PROGRAM P_ADS_1
VAR
	sTextAlarm1				: WSTRING(255);
	sTextAlarm2				: WSTRING(255);
	sTextAlarm3				: WSTRING(255);
	user					: WSTRING(80);
	iNumberAlarm			: INT;
	bTrigger				: BOOL;
	
	fbRead_1: FB_ReadAdsSymByName;
	fbRead_2: FB_ReadAdsSymByName;
	fbRead_3: FB_ReadAdsSymByName;
	fbCyclicReadout: TON;
	fbRead_4: FB_ReadAdsSymByName;
	fbRead_5: FB_ReadAdsSymByName;
	fbLocaltime: FB_LocalSystemTime;

END_VAR

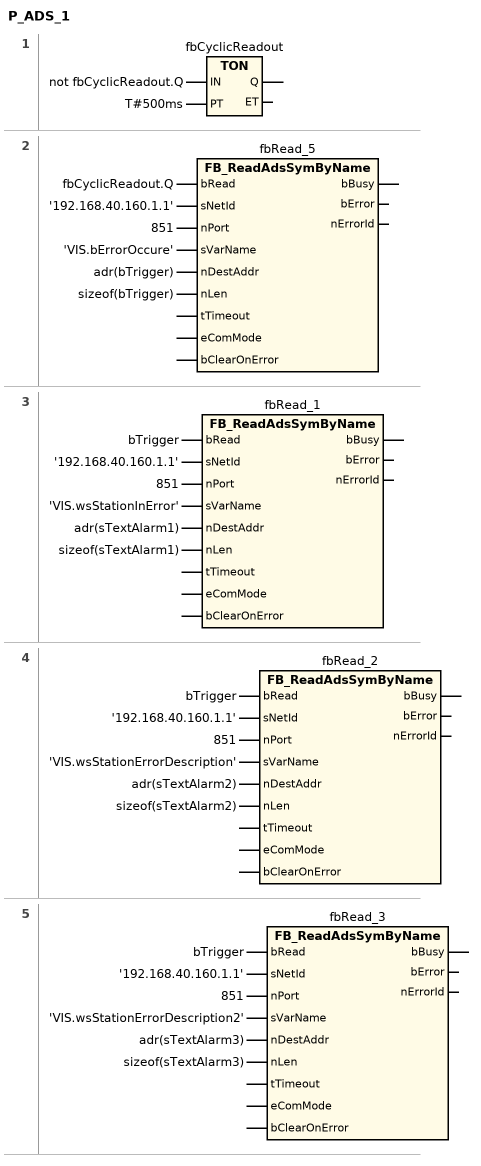
// NETWORK 1
fbCyclicReadout(IN := not fbCyclicReadout.Q, PT := T#500ms); // TON

// NETWORK 2
fbRead_5(
    bRead := fbCyclicReadout.Q,
    sNetId := '192.168.40.160.1.1',
    nPort := 851,
    sVarName := 'VIS.bErrorOccure',
    nDestAddr := adr(bTrigger),
    nLen := sizeof(bTrigger)); // FB_ReadAdsSymByName

// NETWORK 3
fbRead_1(
    bRead := bTrigger,
    sNetId := '192.168.40.160.1.1',
    nPort := 851,
    sVarName := 'VIS.wsStationInError',
    nDestAddr := adr(sTextAlarm1),
    nLen := sizeof(sTextAlarm1)); // FB_ReadAdsSymByName

// NETWORK 4
fbRead_2(
    bRead := bTrigger,
    sNetId := '192.168.40.160.1.1',
    nPort := 851,
    sVarName := 'VIS.wsStationErrorDescription',
    nDestAddr := adr(sTextAlarm2),
    nLen := sizeof(sTextAlarm2)); // FB_ReadAdsSymByName

// NETWORK 5
fbRead_3(
    bRead := bTrigger,
    sNetId := '192.168.40.160.1.1',
    nPort := 851,
    sVarName := 'VIS.wsStationErrorDescription2',
    nDestAddr := adr(sTextAlarm3),
    nLen := sizeof(sTextAlarm3)); // FB_ReadAdsSymByName

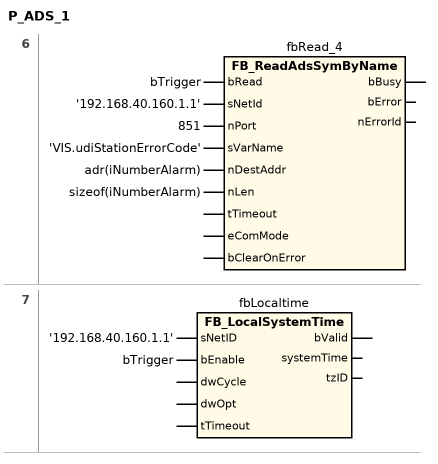
// NETWORK 6
fbRead_4(
    bRead := bTrigger,
    sNetId := '192.168.40.160.1.1',
    nPort := 851,
    sVarName := 'VIS.udiStationErrorCode',
    nDestAddr := adr(iNumberAlarm),
    nLen := sizeof(iNumberAlarm)); // FB_ReadAdsSymByName

// NETWORK 7
fbLocaltime(sNetID := '192.168.40.160.1.1', bEnable := bTrigger); // FB_LocalSystemTime

END_PROGRAM

(* stored: Version 1.1.0.1, ProductVersion 3.1.4024.12
   POU P_ADS_1: Id {6aa95959-5d84-4766-8115-37a607744cea}, SpecialFunc None *)
